TYPE
    ST_HalfAuto_Shipping :
    STRUCT
    END_STRUCT
END_TYPE

(* stored: Version 1.1.0.1, ProductVersion 3.1.4024.13
   DUT ST_HalfAuto_Shipping: Id {adf58bf4-0fbf-40cc-bbb1-b013f60b3445} *)
